TYPE DOutputs :
STRUCT
	output1 : BOOL;
	output2 : BOOL;
	output3 : BOOL;
	output4 : BOOL;
	controlOutput1 : BOOL;
	controlOutput2 : BOOL;
	controlOutput3 : BOOL;
	controlOutput4 : BOOL;
END_STRUCT
END_TYPE

(* stored: Version 1.1.0.1, ProductVersion 3.1.4024.11
   DUT DOutputs: Id {c6c0ae13-0d4b-4c21-9a2f-0c958617c5a6} *)
